// TIA Portal V17 export
// export: Created 2023-04-04T13:27:26.2903614Z, ExportSetting WithDefaults, DisplayName Totally Integrated Automation Portal, DisplayVersion V17, DisplayName TIA Portal Openness, DisplayVersion V17, DisplayName TIA Portal Version Control Interface, DisplayVersion V17, DisplayName STEP 7 Professional, DisplayVersion V17, DisplayName STEP 7 Safety, DisplayVersion V17, DisplayName WinCC Advanced, DisplayVersion V17
DATA_BLOCK "gtyp_SLD"   // DB24
TITLE = Global DB SLD
{ S7_Optimized_Access := 'TRUE' }
AUTHOR : A.Schaefer
VERSION : 0.0
// stored: AutoNumber true, DBAccessibleFromOPCUA true, DBAccessibleFromWebserver true, InstanceOfName typ_SLD, InstanceOfType UDT, IsOnlyStoredInLoadMemory false, IsWriteProtectedInAS false
"typ_SLD"
   // VAR RETAIN
   //    x_Error : Bool;
   //    i_CounterValue_Blue : Int := 26;
   //    i_CounterValue_White : Int := 5;
   //    i_CounterValue_Red : Int := 16;
   //    i_Counter_Actual : Int;
   //    w_Threshold_White_Red : Word := 16#2698;
   //    w_Threshold_Red_Blue : Word := 16#3D41;
   //    Workpiece : "typ_Workpiece";
   //    History { S7_SetPoint := 'True'} : Array[1..20] of "typ_History";
   // END_VAR
BEGIN
END_DATA_BLOCK
